FUNCTION_BLOCK TcLogCore IMPLEMENTS ILogCore
VAR
	{attribute 'hide'} 
	_loggingSingleton : TcLog; // Logger-Singleton: Required to provide Singleton-functionality for TcLog.
	{attribute 'hide'} 			
	_localTimeAsFileTime : Tc2_Utilities.T_FILETIME; // Actual time as filetime, corrected to local time zone
	{attribute 'hide'} 			
	_utcTimeAsFileTime : Tc2_Utilities.T_FILETIME; // Actual time as filetime
	{attribute 'hide'} 
	_timeAsSystemTime : Tc2_Utilities.TIMESTRUCT; // Actual time as timestring
	{attribute 'hide'} 
	_timeAsString : STRING; // Actual time as string
	{attribute 'hide'} 
	_logCache : DynamicStringBuffer; // Dynamic string buffer to cache logs to be processed
	{attribute 'hide'} 
	_startLoggingConfiguration : BOOL; // Aux variable to provide fluent interface.
	{attribute 'hide'} 
	_internalErrorOccured : BOOL; // Aux variable to log internal errors to Error-property.
	{attribute 'hide'}                                                        				
	_config : LoggingConfiguration; // Logging configuration. Is set by invoking configuration methods.
	{attribute 'hide'} 
	_error : Error; // Contains information about internal error.
	{attribute 'hide'} 
	_busy : BOOL; // Logger is busy, typically with writing logs to the file system.
END_VAR

// Nothing to be done here. Logger works by invoking its methods.
// "RunLogger" contains all the implementation that has to be processed cyclically.

// Builds logging configuration.
// Required to provide a fluent interface.
// Has to be called at the begin of each method that configures the logger.
{attribute 'hide'}
METHOD PRIVATE BuildLoggingConfiguration : BOOL
IF NOT _startLoggingConfiguration THEN
	_startLoggingConfiguration := TRUE;
	
	_config.RollingInterval := RollingIntervals.Daily;
	_config.WriteToAds := FALSE;
	_config.FileName := '';
	_config.FilePath := 'c:\';
	_config.MinimumLevel := LogLevels.Debug;
	_config.Delimiter := '|';
	_config.IncludeInstancePath := FALSE;
	_config.LogFileLifespan := 0;
	_config.TimestampFormat := 'YYYYMMDD_hhmm_';
END_IF
END_METHOD

{attribute 'monitoring':='call'}
PROPERTY Busy : BOOL
GET
Busy := _busy;
END_GET
SET // PRIVATE
_busy := Busy;
END_SET
END_PROPERTY

// Returns the current configuration of the logger.
PROPERTY Configuration : LoggingConfiguration
GET
Configuration := _config;
END_GET
END_PROPERTY

// Configuration method.
// Sets the lifespan of log files. Once exceeded, they will be deleted.
METHOD DeleteLogFilesAfterDays : REFERENCE TO TcLogCore
VAR_INPUT
	Lifespan : UINT; // Lifespan of logfiles in days. Once exceeded, log files will be deleted.
END_VAR
BuildLoggingConfiguration();

_config.LogFileLifespan := Lifespan;

DeleteLogFilesAfterDays REF= THIS^;
END_METHOD

// Returns information about internal errors.
{attribute 'monitoring':='call'}
PROPERTY Error : REFERENCE TO Error
GET
Error REF= _error;
END_GET
END_PROPERTY

{attribute 'hide'} 
METHOD FB_init : BOOL
VAR_INPUT
	bInitRetains : BOOL; // if TRUE, the retain variables are initialized (warm start / cold start)
	bInCopyCode : BOOL; // if TRUE, the instance afterwards gets moved into the copy code (online change)
	BufferSize : DINT; // Buffer size for string buffer
END_VAR
_loggingSingleton.Init(THIS^);
_logCache.Init(DINT_TO_UDINT(BufferSize));
END_METHOD

{attribute 'hide'} 
METHOD FB_reinit : BOOL
VAR_INPUT
	BufferSize : DINT; // Buffer size for string buffer
END_VAR
_loggingSingleton.Init(THIS^);
_logCache.Init(DINT_TO_UDINT(BufferSize));
END_METHOD

METHOD FlushCache : BOOL
_logCache.FlushCache();
END_METHOD

// Configuration method.
// Specifies, if instance path should be included in log file.
METHOD IncludeInstancePath : REFERENCE TO TcLogCore
BuildLoggingConfiguration();

_config.IncludeInstancePath := TRUE;

IncludeInstancePath REF= This^;
END_METHOD

// Logger method.
// Logs data in custom format. No additional formatting will be done.
METHOD LogCustomFormat : BOOL
VAR_INPUT
	Data : Tc2_System.T_MaxString; // Data to be logged. No additional formatting will be done.
END_VAR
IF _config.WriteToAds THEN 
	Tc2_System.ADSLOGSTR(ADSLOG_MSGTYPE_LOG OR ADSLOG_MSGTYPE_HINT, Data, ''); 
END_IF

IF _config.FileName <> '' THEN 
	_logCache.AddLine(Data);
END_IF
END_METHOD

// Logger method.
// Logs in the standard format. This includes
// - timestamp
// - log level
// - log message
// - instance path of logging source (optional)
// The message will only be logged if the logging level exceeds the configured minimum logging level.
METHOD LogStandardFormat : BOOL
VAR_INPUT
	Data : Tc2_System.T_MaxString; // Data to be logged. Additional formatting wil be done.
	InstancePath : Tc2_System.T_MaxString; // Instance path of calling logger to locate source of logging message.
	LogLevel : LogLevels; // Log level of message.
END_VAR
VAR_INST
	stringBuilder : StringBuilder;
END_VAR
IF LogLevel >= _config.MinimumLevel THEN
	IF _config.WriteToAds THEN 
		Tc2_System.ADSLOGSTR(
			ADSLOG_MSGTYPE_LOG OR LogLevelToAdsLogMsgType(LogLevel), 
			stringBuilder
				.Reset()
				.AppendIf(_config.IncludeInstancePath, InstancePath)
				.AppendIf(_config.IncludeInstancePath, _config.Delimiter)
				.Append(Data)
				.ToString(), 
			''
		); 
	END_IF
	
	IF _config.FileName <> '' THEN 
		_logCache.AddLine(
			stringBuilder
					.Reset()
					.Append(_timeAsString)
					.Append(_config.Delimiter)
					.Append(TO_STRING(LogLevel))
					.AppendIf(_config.IncludeInstancePath, _config.Delimiter)
					.AppendIf(_config.IncludeInstancePath, InstancePath)
					.Append(_config.Delimiter)
					.Append(Data)
					.ToString()
		);
	END_IF
END_IF
END_METHOD

// Configuration method.
// Sets the minimum log level. Log messages below this level 
// will not be logged.
METHOD MinimumLevel : REFERENCE TO TcLogCore
VAR_INPUT
	Level : LogLevels; // Minimum log level to be logged.
END_VAR
BuildLoggingConfiguration();

_config.MinimumLevel := Level;

MinimumLevel REF=THIS^;
END_METHOD

// Checks the specified rolling interval for the file name.
// Generates new file name if rolling intervall exceeded.
{attribute 'hide'}
METHOD PRIVATE RollingIntervalReached : BOOL
VAR_INPUT
	CurrentUtcTime : Tc2_Utilities.TIMESTRUCT;
	RollingInterval : RollingIntervals;
END_VAR
VAR_INST
	newHour : Tc2_Standard.R_TRIG;
	newDay : Tc2_Standard.R_TRIG;
	newMonth : Tc2_Standard.R_TRIG;
	
	hourRolled : BOOL;
	dayRolled : BOOL;
	monthRolled : BOOL;
END_VAR
newHour(CLK := (CurrentUtcTime.wMinute = 0 AND CurrentUtcTime.wSecond = 0), 
	Q => hourRolled);
newDay(CLK := (hourRolled AND CurrentUtcTime.wHour = 0), 
	Q => dayRolled);
newMonth(CLK := (dayRolled AND CurrentUtcTime.wDay = 1), 
	Q => monthRolled);

RollingIntervalReached := 	(hourRolled 	AND RollingInterval = RollingIntervals.Hourly) OR
							(dayRolled 		AND RollingInterval = RollingIntervals.Daily) 	OR
							(monthRolled 	AND RollingInterval = RollingIntervals.Monthly);
END_METHOD

// Cyclic method of Logger.
// This method has to be executed in every plc cycle and runs 
// all internal methods that have to be executed cyclically.
METHOD RunLogger : BOOL
VAR_INST
	newDay : Tc2_Standard.R_TRIG; 
	dateTime : DateTime;
	deleteExpiredLogFiles : DeleteOldFiles;
	fileNameStringBuilder : StringBuilder;
	timeStamp : STRING; // Timestamp used for filename
END_VAR
// Generate time data (shared state)
dateTime();
	
_localTimeAsFileTime := dateTime.AsLocalFileTime;
_timeAsSystemTime := dateTime.AsLocalSystemTime;
_timeAsString := dateTime.AsLocalSystemTimeString;

// Generate new timestamp for filename
IF RollingIntervalReached(_timeAsSystemTime, _config.RollingInterval) OR dateTime.Done THEN
	timeStamp := dateTime.ToFormatString(_config.TimestampFormat);
END_IF

// Delete expired log files
newDay(CLK := _timeAsSystemTime.wHour = 0);
deleteExpiredLogFiles(
	StartScan 			:= 	newDay.Q AND (_config.LogFileLifespan > 0),
	ExpirationInDays 	:=	_config.LogFileLifespan,
	FilePath			:=	_config.FilePath,
	FileName 			:=	_config.FileName,
	CurrentUtcTime 		:= 	_utcTimeAsFileTime	
	);
IF deleteExpiredLogFiles.Error.Active THEN
	_internalErrorOccured := TRUE;
	_error := deleteExpiredLogFiles.Error;
END_IF
		
// Persist logging messages to file
_logCache.PersistToFile(
	fileNameStringBuilder
		.Reset()
		.Append(_config.FilePath)
		.AppendIf(Tc2_Standard.RIGHT(_config.FilePath, 1) <> '\', '\')
		.Append(timeStamp)
		.Append(_config.FileName)
		.ToString()
);
IF _logCache.Error.Active THEN
	_internalErrorOccured := TRUE;
	_error := _logCache.Error;
END_IF

// Forward busy state of LogCache 
Busy := _logCache.Busy;

// Reset Logging configuration: neccesary in order to provide fluent interface
_startLoggingConfiguration := FALSE;

// Reset error flag each cycle to automatically confirm errors once they are gone.
IF NOT _internalErrorOccured THEN
	_error.Active := FALSE;
	_error.Code := ErrorCodes.None;
	_error.Info := '';
END_IF
_internalErrorOccured := FALSE;
END_METHOD

// Configuration method
// Sets delimiter between different columns of log file.
METHOD SetDelimiter : REFERENCE TO TcLogCore
VAR_INPUT
	Delimiter : STRING(1); // Delimiter between different columns of log file.
END_VAR
BuildLoggingConfiguration();

_config.Delimiter := Delimiter;

SetDelimiter REF=THIS^;
END_METHOD

// Configuration method
// Sets the rolling interval of the log file. Once the rolling interval
// expires, a file name with a new timestamp will be generated.
METHOD SetRollingInterval : REFERENCE TO TcLogCore
VAR_INPUT
	Interval : RollingIntervals; // Rolling interval for log file. Once exceeded, a new log file will be created.
END_VAR
BuildLoggingConfiguration();

_config.RollingInterval := Interval;

SetRollingInterval REF= THIS^;
END_METHOD

// Configuration method
// Sets the format of the timestamp in the file name.
METHOD TimestampFormat : REFERENCE TO TcLogCore
VAR_INPUT
	Format : STRING; // Format the timestamp should have
END_VAR
BuildLoggingConfiguration();

_config.TimestampFormat := Format;

TimestampFormat REF= THIS^;
END_METHOD

// Configuration method.
// Writes logdata to ADS log.
METHOD WriteToAds : REFERENCE TO TcLogCore
BuildLoggingConfiguration();

_config.WriteToAds := TRUE;

WriteToAds REF= This^;
END_METHOD

// Configuration method.
// Writes log message to file.
METHOD WriteToFile : REFERENCE TO TcLogCore
VAR_INPUT
	Path : Tc2_System.T_MaxString; // File path to be written to. Has to end with '\'.
	FileName : STRING; // File name to be written to. Will automatically be prefixed by timestamp.
END_VAR
BuildLoggingConfiguration();

_config.FilePath := Path;
_config.FileName := FileName;

WriteToFile REF= This^;
END_METHOD

END_FUNCTION_BLOCK

(* stored: Version 1.1.0.1
   POU TcLogCore: Id {81f82071-4a6c-4f57-9a56-0ade3c0c9c94}, SpecialFunc None
   Method BuildLoggingConfiguration: Id {eddda5b2-7aed-4925-82c6-d1cc02972392}
   Property Busy: Id {2506cebb-3f61-4c95-90db-f0f540dd9e98}
   Get Get: Id {addca3d4-1294-4daf-817b-bf0ea7026f56}
   Set Set: Id {75c50778-a1c9-4233-8355-44379e5bd491}
   Property Configuration: Id {05d13daa-5623-41b4-ae7a-41103edd188e}
   Get Get: Id {7fd81f24-ea07-4e82-8550-f6e8c4f01f6e}
   Method DeleteLogFilesAfterDays: Id {474486bd-99ed-4f8f-b78b-4c4c8ea5cfc8}
   Property Error: Id {6fb536cf-61ab-4968-94e7-6a0e9727441d}
   Get Get: Id {8cae9ed2-7297-4ac6-8c06-f53f0a38a91c}
   Method FB_init: Id {2d60871a-4b97-4f7f-9afb-379a9cace715}
   Method FB_reinit: Id {7a4a2895-bc8f-4c5f-ae34-d121f2978f2a}
   Method FlushCache: Id {d85421f8-abe8-45dc-a84c-3e5e5c8a80e5}
   Method IncludeInstancePath: Id {a3af0de9-912d-4997-ab67-451214c74322}
   Method LogCustomFormat: Id {b807e7a1-f0a7-4c3d-8d69-25482e8e77ab}
   Method LogStandardFormat: Id {4daf0b25-d1e4-454d-aade-383a8ce5cffd}
   Method MinimumLevel: Id {2c064562-d9e7-47af-9d8e-602f3edf874f}
   Method RollingIntervalReached: Id {46ff7d34-a17e-4357-ab5f-b5dd39bd8821}
   Method RunLogger: Id {46efeb58-43e6-49ca-b3ab-11723675a9a3}
   Method SetDelimiter: Id {dc4c96e1-55b5-4273-91d7-557c2f84a7f0}
   Method SetRollingInterval: Id {ccb17be1-b0a9-460e-b8ac-cfc6fa396397}
   Method TimestampFormat: Id {ae9acdda-63d0-4143-b862-4bb5f08b434d}
   Method WriteToAds: Id {0ac63c1b-765b-40a5-b132-bcc3d18f2f34}
   Method WriteToFile: Id {c27c86ab-078c-40d8-8991-697cd72b869c} *)
